(* IEC 61131-3 sources: OMJSON/src/Ar/Lux/LuxProg, 1 file *)

(* ---- Main.st ---- *)
(*
* File: Main.st
* Copyright (c) 2023 Loupe
* https://loupe.team
*
* This file is part of OMJSON, licensed under the MIT License.
*)

// This program serves variables to web applications via WebSockets and
// a JSON interface

PROGRAM _INIT

    // pCache is required
	jsonWebSocketServer_0.pCacheArray := ADR(jsonCache);
	jsonWebSocketServer_0.maxClients := MAX_CLIENTS;

	// Note: ServerIP, ServerPort, BufferSize, and MaxIterations are optional and not set
	// Without a ServerIP the server listens on all ethernet interfaces.
	// Set ServerIP to the address of the interface the HMI is connected to if the PLC has more than one
	jsonWebSocketServer_0.BufferSize := 200000;

	gLuxAccess.pEntries := ADR(gLuxAccessList);
	gLuxAccess.numEntries := LUX_MAI_ACCESS + 1;

	// Call jsonWebSocketServer once in the INIT routine to allocate internal memory
	jsonWebSocketServer_0();

END_PROGRAM

PROGRAM _CYCLIC

	// Restrict clients to the variables in gLuxAccessList as soon as the application fills it.
	// This is checked cyclically because the application's INIT might run after this one.
	// While the list is empty clients can read and write ALL variables (jsonWebSocketServer_0.AccessControlActive = FALSE)
	IF gLuxAccessList[0].name <> '' THEN
		jsonWebSocketServer_0.pAccess := ADR(gLuxAccess);
	END_IF

	// Call jsonWebSocketServer cyclically to serve variables
	jsonWebSocketServer_0();

	IF NOT SimulationStatus(0) THEN
		gWSTimeout := FALSE;
		FOR i:=0 TO JSON_MAI_CLIENTS DO
			// On any client disconnect
			IF oldClientInfo[i].Connected AND NOT jsonWebSocketServer_0.ClientInfo[i].Connected THEN
				gWSTimeout := TRUE;
			END_IF
		END_FOR
		oldClientInfo := jsonWebSocketServer_0.ClientInfo;
	END_IF

END_PROGRAM
